// TIA Portal V19 export
DATA_BLOCK "A0302_Manipolatore"   // DB117
// stored: InstanceOfName A0302_Manipolatore_FB, InstanceOfType FB
"A0302_Manipolatore_FB"
   // VAR_INPUT
   //    AreaInterface : "AreaInterface";
   //    ZSI : "udt_ZoneSafetyInterface";
   //    DSI_Testa_Feed : "udt_DeviceSafetyInterface";
   //    DSI_Coda_Feed : "udt_DeviceSafetyInterface";
   //    DSI_Valve : "udt_DeviceSafetyInterface";
   //    Drive_Testa : "TAx_DriveInterface";
   //    Drive_Coda : "TAx_DriveInterface";
   //    DataIn : Struct
   //       OP_MoveToPos : Bool;
   //       Sollevamento : Struct
   //          OP : "OP_PB";
   //       END_STRUCT;
   //       Magneti : Struct
   //          OP : "OP_PB";
   //       END_STRUCT;
   //       Sens : Struct
   //          Ls1 : Bool;
   //          Ls2 : Bool;
   //          Ls3 : Bool;
   //          Ls4 : Bool;
   //       END_STRUCT;
   //    END_STRUCT;
   //    CIn : Struct
   //       Manager : Struct
   //          EnableStopDoorOpeningReq { ExternalAccessible := 'False'; ExternalVisible := 'False'; ExternalWritable := 'False'} : Bool;
   //          EnableStopInPhase { ExternalAccessible := 'False'; ExternalVisible := 'False'; ExternalWritable := 'False'} : Bool;
   //          EnableStopProgrammed { ExternalAccessible := 'False'; ExternalVisible := 'False'; ExternalWritable := 'False'} : Bool;
   //          Control_ON { ExternalAccessible := 'False'; ExternalVisible := 'False'; ExternalWritable := 'False'} : Bool;
   //          MoveToPos { ExternalAccessible := 'False'; ExternalVisible := 'False'; ExternalWritable := 'False'} : Bool;
   //          Pos { ExternalAccessible := 'False'; ExternalVisible := 'False'; ExternalWritable := 'False'} : LReal;
   //          Vel : LReal;
   //          Acc : LReal;
   //          Dec : LReal;
   //          Sollevamento { ExternalAccessible := 'False'; ExternalVisible := 'False'; ExternalWritable := 'False'} : Struct
   //             Rest : Bool;
   //             Work : Bool;
   //          END_STRUCT;
   //          Magneti { ExternalAccessible := 'False'; ExternalVisible := 'False'; ExternalWritable := 'False'} : Struct
   //             Rest : Bool;
   //             Work : Bool;
   //          END_STRUCT;
   //       END_STRUCT;
   //       OP_SemiAut_PB { ExternalWritable := 'False'} : Bool;
   //       Rulliera { ExternalWritable := 'False'} : Struct
   //          Centratori : "ValveMachine_COut";
   //          Coda : Struct
   //             Sens : Struct
   //                FTC_Rall : Bool;
   //                FTC_Prox_Ing : Bool;
   //             END_STRUCT;
   //          END_STRUCT;
   //          Centro : Struct
   //             Sens : Struct
   //                FTC_Centrale : Bool;
   //             END_STRUCT;
   //          END_STRUCT;
   //       END_STRUCT;
   //       CarroPareggTesta { ExternalWritable := 'False'} : Struct
   //          Sens : Struct
   //             FTC1_Rall : Bool;
   //             FTC2_Prox_Ls : Bool;
   //             PresenzaMat : Bool;
   //          END_STRUCT;
   //       END_STRUCT;
   //       CarroPareggCoda { ExternalWritable := 'False'} : Struct
   //          Sens : Struct
   //             FTC_Ingombro_In : Bool;
   //             FTC_Ingombro_Out : Bool;
   //             PresenzaMat : Bool;
   //          END_STRUCT;
   //       END_STRUCT;
   //       CarriPareggiatori : Struct
   //          ZoneA0302Entry_Empty { ExternalWritable := 'False'} : Bool;
   //          ZoneA0302Exit_Empty { ExternalWritable := 'False'} : Bool;
   //          RequestNewPosition : Bool;
   //       END_STRUCT;
   //       Spalle : Struct
   //          Coda : Struct
   //             ActualPos : LReal;
   //          END_STRUCT;
   //          Testa : Struct
   //             ActualPos : LReal;
   //          END_STRUCT;
   //       END_STRUCT;
   //    END_STRUCT;
   //    Config : Struct
   //       Testa : Struct
   //          Ax : "Positioning_EPOS_Machine_Config_NEW";
   //          Sollevatore : "ValveMachine_Config";
   //          Magnete : "ValveMachine_Config";
   //       END_STRUCT;
   //       Coda : Struct
   //          Ax : "Positioning_EPOS_Machine_Config_NEW";
   //          Sollevatore : "ValveMachine_Config";
   //          Magnete : "ValveMachine_Config";
   //       END_STRUCT;
   //       DelayMissingCondition : Time;
   //    END_STRUCT;
   //    HWID_AxTesta_TEL111 : HW_SUBMODULE;
   //    HWID_AxCoda_TEL111 : HW_SUBMODULE;
   // END_VAR
   // VAR_OUTPUT
   //    MachineInterface : "MachineInterface";
   //    COut : Struct
   //       Testa : Struct
   //          Ax : "Positioning_EPOS_Machine_COut";
   //          Sollevatore : "ValveMachine_COut";
   //          Magnete : "ValveMachine_COut";
   //       END_STRUCT;
   //       Coda : Struct
   //          Ax : "Positioning_EPOS_Machine_COut";
   //          Sollevatore : "ValveMachine_COut";
   //          Magnete : "ValveMachine_COut";
   //       END_STRUCT;
   //       CheckAxTesta : Struct
   //          InPos_Prelievo : Bool;
   //          InPos_BancoScarto : Bool;
   //          InPos_BancoA0303 : Bool;
   //       END_STRUCT;
   //       CheckAxCoda : Struct
   //          InPos_Prelievo : Bool;
   //          InPos_BancoScarto : Bool;
   //          InPos_BancoA0303 : Bool;
   //       END_STRUCT;
   //       InPos_Prelievo : Bool;
   //       InPos_BancoScarto : Bool;
   //       InPos_BancoA0303 : Bool;
   //       OutWorkSpace : Bool;
   //    END_STRUCT;
   // END_VAR
   // VAR_IN_OUT
   //    Par : Struct
   //       Ax : "Positioning_EPOS_Machine_Par";
   //       Ax_Aut : "A0301_Mach_Speed_Par";
   //       Ax_Pos : Struct
   //          Prelievo : LReal;
   //          BancoCtrl : LReal;
   //          BancoA0303 : LReal;
   //          Tollerance : Struct
   //             Prelievo : LReal;
   //             BancoCtrl : LReal;
   //             BancoA0303 : LReal;
   //          END_STRUCT;
   //       END_STRUCT;
   //    END_STRUCT;
   //    Pers_Data : Struct
   //       EncoderAbsolute_Preset_OK : Bool;
   //       Persistent_ActualPosition : LReal;
   //    END_STRUCT;
   // END_VAR
   // VAR
   //    Alarm : Struct
   //       Testa : Struct
   //          Ax : "Positioning_EPOS_Machine_Alr";
   //          Sollevatore : "ValveAlr";
   //          Magnete : "ValveAlr";
   //       END_STRUCT;
   //       Coda : Struct
   //          Ax : "Positioning_EPOS_Machine_Alr";
   //          Sollevatore : "ValveAlr";
   //          Magnete : "ValveAlr";
   //       END_STRUCT;
   //       CheckBothAxMove : Bool;
   //    END_STRUCT;
   //    Warning : Struct
   //       Testa : Struct
   //          Ax : "Positioning_EPOS_Machine_Wng";
   //          Sollevatore : "ValveMachine_Wng";
   //          Magnete : "ValveMachine_Wng";
   //       END_STRUCT;
   //       Coda : Struct
   //          Ax : "Positioning_EPOS_Machine_Wng";
   //          Sollevatore : "ValveMachine_Wng";
   //          Magnete : "ValveMachine_Wng";
   //       END_STRUCT;
   //       MissingCnd : Struct
   //          OP_REST_Sollevamento : Bool;
   //          OP_WORK_Sollevamento : Bool;
   //          OP_REST_Magneti : Bool;
   //          OP_WORK_Magneti : Bool;
   //       END_STRUCT;
   //    END_STRUCT;
   //    HMI : Struct
   //       Selection : Struct
   //          Ax : Int;
   //       END_STRUCT;
   //       Ax_Testa : "AnalogSens_HmiData";
   //       Ax_Coda : "AnalogSens_HmiData";
   //    END_STRUCT;
   //    Sts : Struct
   //       ReadyForMove : Bool;
   //       OP_Manip_CanMoveFreely : Bool;
   //       OP_Ax_CanMoveFreely : Bool;
   //       Op_MoveToPos_Cnd : Bool;
   //       Sollevamento : Struct
   //          OP_Rest_Cnd : Bool;
   //          Op_Work_Cnd : Bool;
   //       END_STRUCT;
   //       Magneti : Struct
   //          OP_Rest_Cnd : Bool;
   //          Op_Work_Cnd : Bool;
   //       END_STRUCT;
   //       Coda_PermessoDaSynchOk : Bool;
   //       Testa_PermessoDaSynchOk : Bool;
   //    END_STRUCT;
   //    Ctrl : Struct
   //       Sollevamento : Struct
   //          OP_Rest_Man : Bool;
   //          OP_Work_Man : Bool;
   //          OP_Rest_Aut : Bool;
   //          OP_Work_Aut : Bool;
   //          OP_Rest : Bool;
   //          OP_Work : Bool;
   //       END_STRUCT;
   //       Magneti : Struct
   //          OP_Rest_Aut : Bool;
   //          OP_Work_Aut : Bool;
   //          OP_Rest_Man : Bool;
   //          OP_Work_Man : Bool;
   //          OP_Rest : Bool;
   //          OP_Work : Bool;
   //       END_STRUCT;
   //       Ax : Struct
   //          OP_MoveToPos_Man : Bool;
   //          OP_MoveToPos_Aut : Bool;
   //          OP_MoveToPos : Bool;
   //       END_STRUCT;
   //    END_STRUCT;
   //    AUX : Struct
   //       OP_MoveToPos : Bool;
   //       Sollevamento : Struct
   //          OP_Rest : Bool;
   //          OP_Work : Bool;
   //       END_STRUCT;
   //       Magneti : Struct
   //          OP_Rest : Bool;
   //          OP_Work : Bool;
   //       END_STRUCT;
   //    END_STRUCT;
   //    Ax_Testa : "Positioning_EPOS_Machine_FB_NEW";
   //    Ax_Coda : "Positioning_EPOS_Machine_FB_NEW";
   //    Sollevatore_Testa { S7_SetPoint := 'True'} : "ValveMachine_FB";
   //    Sollevatore_Coda { S7_SetPoint := 'True'} : "ValveMachine_FB";
   //    Magnete_Testa { S7_SetPoint := 'True'} : "ValveMachine_FB";
   //    Magnete_Coda { S7_SetPoint := 'True'} : "ValveMachine_FB";
   //    TON_Magneti : Struct
   //       OP_REST_MissingCnd { S7_SetPoint := 'True'} : TON_TIME;
   //       OP_WORK_MissingCnd { S7_SetPoint := 'True'} : TON_TIME;
   //    END_STRUCT;
   //    TON_Sollevamento : Struct
   //       OP_REST_MissingCnd { S7_SetPoint := 'True'} : TON_TIME;
   //       OP_WORK_MissingCnd { S7_SetPoint := 'True'} : TON_TIME;
   //    END_STRUCT;
   //    TON_CheckAxMove : IEC_TIMER;
   //    CheckAxisSynch { ExternalAccessible := 'False'; ExternalVisible := 'False'; ExternalWritable := 'False'} : "CheckAxisSynch";
   //    Sts_PosAxis { S7_SetPoint := 'True'} : Int;
   // END_VAR
BEGIN
END_DATA_BLOCK
